// SIMATIC S7-200 project (STEP 7-Micro/WIN), CPU 224XP REL 02.01

SYMBOL_TABLE USUARIO1
PMARCHA          I0.0     // PULASADOR DR MARCHA
FC_ABAJO         I0.1     // FC GANCHO ABAJO
FC_ARRIBA        I0.2     // FC GANCHO ARRIBA
FC_IZQUIERDA     I0.3     // FC IZQUIERDA
FC_TANQUE_1      I0.4     // FC TANQUE 1
FC_TANQUE_2      I0.5     // FC TANQUE 2
FC_TANQUE_3      I0.6     // FC TANQUE 3
SUBIR            Q0.0     // SUBIDA GANCHO
BAJAR            Q0.1     // BAJADA GANCHO
derecha          Q0.2     // DESPLAZAMIENTO CARRO IZQUIERDA
izquierda        Q0.3     // DESPLAZAMIENTO CARRO DERECHA
subir_control    M0.0
bajar_control    M0.1
derechacontrol   M0.2
izquierdacontrol M0.3
END_SYMBOL_TABLE

ORGANIZATION_BLOCK PRINCIPAL:OB1
TITLE=GRUA PROCESO VULNERABLE A LA OXIDACION
// 
BEGIN
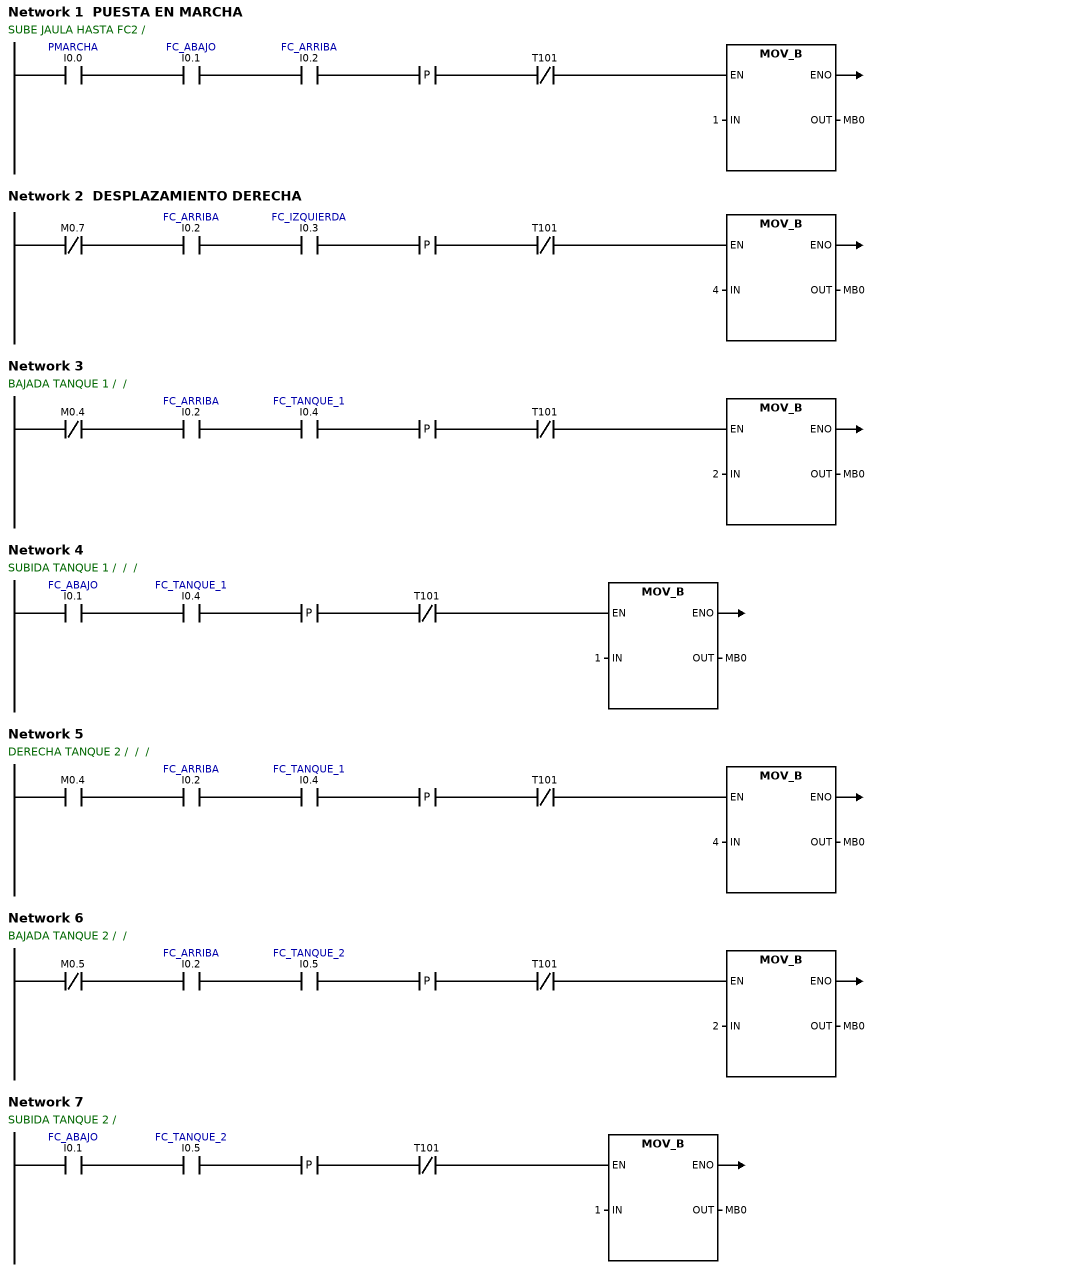
Network 1 // PUESTA EN MARCHA

// SUBE JAULA HASTA FC2
// 
LD     PMARCHA:I0.0
A      FC_ABAJO:I0.1
A      FC_ARRIBA:I0.2
EU
AN     T101
MOVB   1, MB0
Network 2 // DESPLAZAMIENTO DERECHA

LDN    M0.7
A      FC_ARRIBA:I0.2
A      FC_IZQUIERDA:I0.3
EU
AN     T101
MOVB   4, MB0
Network 3
// BAJADA TANQUE 1
// 
// 
LDN    M0.4
A      FC_ARRIBA:I0.2
A      FC_TANQUE_1:I0.4
EU
AN     T101
MOVB   2, MB0
Network 4
// SUBIDA TANQUE 1
// 
// 
// 
LD     FC_ABAJO:I0.1
A      FC_TANQUE_1:I0.4
EU
AN     T101
MOVB   1, MB0
Network 5
// DERECHA TANQUE 2
// 
// 
// 
LD     M0.4
A      FC_ARRIBA:I0.2
A      FC_TANQUE_1:I0.4
EU
AN     T101
MOVB   4, MB0
Network 6
// BAJADA TANQUE 2
// 
// 
LDN    M0.5
A      FC_ARRIBA:I0.2
A      FC_TANQUE_2:I0.5
EU
AN     T101
MOVB   2, MB0
Network 7
// SUBIDA TANQUE 2
// 
LD     FC_ABAJO:I0.1
A      FC_TANQUE_2:I0.5
EU
AN     T101
MOVB   1, MB0
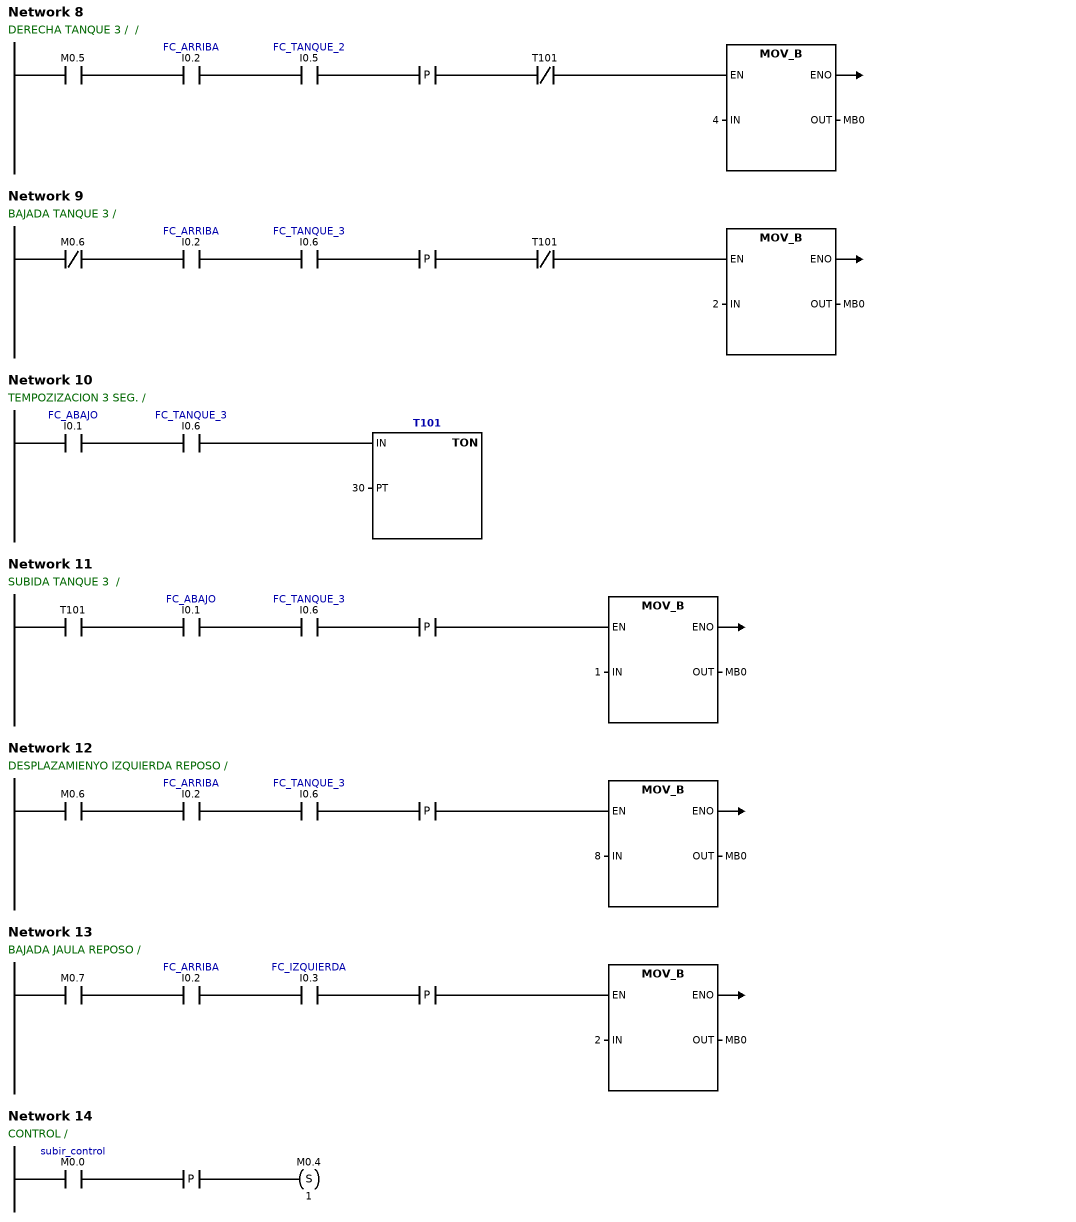
Network 8
// DERECHA TANQUE 3
// 
// 
LD     M0.5
A      FC_ARRIBA:I0.2
A      FC_TANQUE_2:I0.5
EU
AN     T101
MOVB   4, MB0
Network 9
// BAJADA TANQUE 3
// 
LDN    M0.6
A      FC_ARRIBA:I0.2
A      FC_TANQUE_3:I0.6
EU
AN     T101
MOVB   2, MB0
Network 10
// TEMPOZIZACION 3 SEG.
// 
LD     FC_ABAJO:I0.1
A      FC_TANQUE_3:I0.6
TON    T101, 30
Network 11
// SUBIDA TANQUE 3 
// 
LD     T101
A      FC_ABAJO:I0.1
A      FC_TANQUE_3:I0.6
EU
MOVB   1, MB0
Network 12
// DESPLAZAMIENYO IZQUIERDA REPOSO
// 
LD     M0.6
A      FC_ARRIBA:I0.2
A      FC_TANQUE_3:I0.6
EU
MOVB   8, MB0
Network 13
// BAJADA JAULA REPOSO
// 
LD     M0.7
A      FC_ARRIBA:I0.2
A      FC_IZQUIERDA:I0.3
EU
MOVB   2, MB0
Network 14
// CONTROL
// 
LD     subir_control:M0.0
EU
S      M0.4, 1
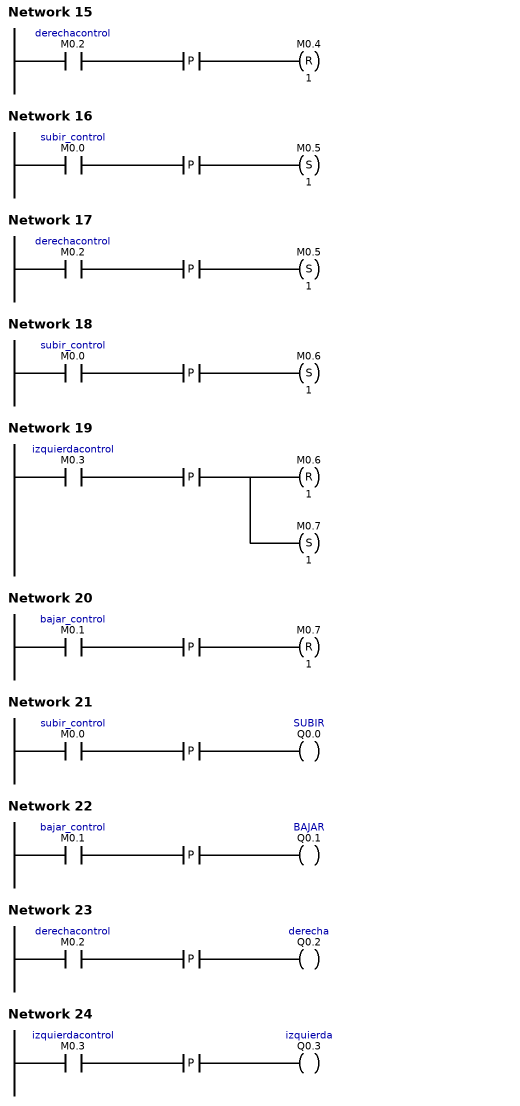
Network 15
LD     derechacontrol:M0.2
EU
R      M0.4, 1
Network 16
LD     subir_control:M0.0
EU
S      M0.5, 1
Network 17
LD     derechacontrol:M0.2
EU
S      M0.5, 1
Network 18
LD     subir_control:M0.0
EU
S      M0.6, 1
Network 19
LD     izquierdacontrol:M0.3
EU
R      M0.6, 1
S      M0.7, 1
Network 20
LD     bajar_control:M0.1
EU
R      M0.7, 1
Network 21
LD     subir_control:M0.0
EU
=      SUBIR:Q0.0
Network 22
LD     bajar_control:M0.1
EU
=      BAJAR:Q0.1
Network 23
LD     derechacontrol:M0.2
EU
=      derecha:Q0.2
Network 24
LD     izquierdacontrol:M0.3
EU
=      izquierda:Q0.3
END_ORGANIZATION_BLOCK
